// TIA Portal V15.1 export
// export: Created 2024-06-21T08:41:12.1834581Z, ExportSetting WithDefaults, DisplayName Totally Integrated Automation Portal, DisplayVersion V15.1 Update 5, DisplayName TIA Portal Openness, DisplayVersion V15.1 Update 5, DisplayName SINAMICS Startdrive Advanced, DisplayVersion V15.1, DisplayName G130, G150, S120, S150, SINAMICS MV, S210, DisplayVersion V15.1, DisplayName G110M, G120, G120C, G120D, G120P, DisplayVersion V15.1, DisplayName STEP 7 Professional, DisplayVersion V15.1 Update 5, DisplayName STEP 7 Safety, DisplayVersion V15.1, DisplayName WinCC Professional, DisplayVersion V15.1 Update 5, DisplayName SIMATIC Visualization Architect, DisplayVersion V15.1
FUNCTION_BLOCK "LGBShiftRegLineSub"   // FB6705, SCL
TITLE = 'L_ShiftRegLineGC'
{ S7_Optimized_Access := 'TRUE' }
VERSION : 0.1
// Block Parameters
// stored: AutoNumber false, IsIECCheckEnabled false, IsRetainMemResEnabled false, MemoryReserve 100, SetENOAutomatically False, UDAEnableTagReadback false
   VAR_INPUT
      I_VEMData { ExternalAccessible := 'False'; ExternalVisible := 'False'; ExternalWritable := 'False'} : "VEMData";   // VEMData
      I_EncPlsCntr { ExternalAccessible := 'False'; ExternalVisible := 'False'; ExternalWritable := 'False'} : DInt;   // Encoder pulse counter - value from counter card
      I_LineRunning { ExternalAccessible := 'False'; ExternalVisible := 'False'; ExternalWritable := 'False'} : Bool;   // Line running - signal from freq. convertor
      I_TriggerDet { ExternalAccessible := 'False'; ExternalVisible := 'False'; ExternalWritable := 'False'} : Bool;   // Trigger sensor
   END_VAR
   VAR_OUTPUT
      O_SetpBodyPitch { ExternalAccessible := 'False'; ExternalVisible := 'False'; ExternalWritable := 'False'} : Int;   // Setpoint Body pitch (cm)
      O_SetpCycleTime { ExternalAccessible := 'False'; ExternalVisible := 'False'; ExternalWritable := 'False'} : Int;   // Setpoint Cycle time (sec)
      O_SetpSpeed { ExternalAccessible := 'False'; ExternalVisible := 'False'; ExternalWritable := 'False'} : Real;   // Setpoint Speed (m/min)
      O_LineIsEmpty { ExternalAccessible := 'False'; ExternalVisible := 'False'; ExternalWritable := 'False'} : Bool;   // Line is empty
      O_AA_EncoderMinMax { ExternalAccessible := 'False'; ExternalVisible := 'False'; ExternalWritable := 'False'} : Bool;   // Settings Min. and Max. range for the encoder is not ok --- Max. must be > Min. and Max. <> 0
      O_AA_SetpointBodyPitch { ExternalAccessible := 'False'; ExternalVisible := 'False'; ExternalWritable := 'False'} : Bool;   // Setpoint Bodypitch is not ok --- Setpoint must be > 100 cm
      O_AA_SetpointCycleTime { ExternalAccessible := 'False'; ExternalVisible := 'False'; ExternalWritable := 'False'} : Bool;   // Setpoint CycleTime is not ok --- Setpoint must be > 10 sec
      O_AA_NbrOfWorkZones { ExternalAccessible := 'False'; ExternalVisible := 'False'; ExternalWritable := 'False'} : Bool;   // Number of work zones is not ok --- Must be >= 2 and <= 30
      O_AA_EncoderPuls { ExternalAccessible := 'False'; ExternalVisible := 'False'; ExternalWritable := 'False'} : Bool;   // The line is running buth there are no encoder pulses
      O_AC_Calibration { ExternalAccessible := 'False'; ExternalVisible := 'False'; ExternalWritable := 'False'} : Bool;   // Calibration is not ok. Let the line run and start the calibration
      O_AC_Area1 { ExternalAccessible := 'False'; ExternalVisible := 'False'; ExternalWritable := 'False'} : Bool;   // Start or End value is not ok
      O_AC_Area2 { ExternalAccessible := 'False'; ExternalVisible := 'False'; ExternalWritable := 'False'} : Bool;   // Start or End value is not ok
      O_AC_Area3 { ExternalAccessible := 'False'; ExternalVisible := 'False'; ExternalWritable := 'False'} : Bool;   // Start or End value is not ok
      O_AC_Area4 { ExternalAccessible := 'False'; ExternalVisible := 'False'; ExternalWritable := 'False'} : Bool;   // Start or End value is not ok
      O_AC_Area5 { ExternalAccessible := 'False'; ExternalVisible := 'False'; ExternalWritable := 'False'} : Bool;   // Start or End value is not ok
      O_AC_Area6 { ExternalAccessible := 'False'; ExternalVisible := 'False'; ExternalWritable := 'False'} : Bool;   // Start or End value is not ok
      O_AC_Area7 { ExternalAccessible := 'False'; ExternalVisible := 'False'; ExternalWritable := 'False'} : Bool;   // Start or End value is not ok
      O_AC_Area8 { ExternalAccessible := 'False'; ExternalVisible := 'False'; ExternalWritable := 'False'} : Bool;   // Start or End value is not ok
      O_AC_Area9 { ExternalAccessible := 'False'; ExternalVisible := 'False'; ExternalWritable := 'False'} : Bool;   // Start or End value is not ok
      O_AC_Area10 { ExternalAccessible := 'False'; ExternalVisible := 'False'; ExternalWritable := 'False'} : Bool;   // Start or End value is not ok
      O_Area1 { ExternalAccessible := 'False'; ExternalVisible := 'False'; ExternalWritable := 'False'} : Bool;   // Position active in the Area
      O_Area2 { ExternalAccessible := 'False'; ExternalVisible := 'False'; ExternalWritable := 'False'} : Bool;   // Position active in the Area
      O_Area3 { ExternalAccessible := 'False'; ExternalVisible := 'False'; ExternalWritable := 'False'} : Bool;   // Position active in the Area
      O_Area4 { ExternalAccessible := 'False'; ExternalVisible := 'False'; ExternalWritable := 'False'} : Bool;   // Position active in the Area
      O_Area5 { ExternalAccessible := 'False'; ExternalVisible := 'False'; ExternalWritable := 'False'} : Bool;   // Position active in the Area
      O_Area6 { ExternalAccessible := 'False'; ExternalVisible := 'False'; ExternalWritable := 'False'} : Bool;   // Position active in the Area
      O_Area7 { ExternalAccessible := 'False'; ExternalVisible := 'False'; ExternalWritable := 'False'} : Bool;   // Position active in the Area
      O_Area8 { ExternalAccessible := 'False'; ExternalVisible := 'False'; ExternalWritable := 'False'} : Bool;   // Position active in the Area
      O_Area9 { ExternalAccessible := 'False'; ExternalVisible := 'False'; ExternalWritable := 'False'} : Bool;   // Position active in the Area
      O_Area10 { ExternalAccessible := 'False'; ExternalVisible := 'False'; ExternalWritable := 'False'} : Bool;   // Position active in the Area
   END_VAR
   VAR_IN_OUT
      IO_ShiftRegData : "ShiftRegData";   // Line data
      IO_Modes : "Modes";   // Modes
      H_HMI : "H_HMI";   // Animation
      H_GBShiftRegLine : "H_GBShiftRegLine";   // Animation
      C_Config : "ShiftRegLineConfig";   // Config
   END_VAR
   VAR
      AlarmEncoderMinMax { ExternalAccessible := 'False'; ExternalVisible := 'False'; ExternalWritable := 'False'} : Bool;   // Settings Min. and Max. range for the encoder is not ok --- Max. must be > Min. and Max. <> 0
      AlarmSetpointBodyPitch { ExternalAccessible := 'False'; ExternalVisible := 'False'; ExternalWritable := 'False'} : Bool;   // Setpoint Bodypitch is not ok --- Setpoint must be > 100 cm
      AlarmSetpointCycleTime { ExternalAccessible := 'False'; ExternalVisible := 'False'; ExternalWritable := 'False'} : Bool;   // Setpoint CycleTime is not ok --- Setpoint must be > 10 sec
      AlarmNbrOfWorkZones { ExternalAccessible := 'False'; ExternalVisible := 'False'; ExternalWritable := 'False'} : Bool;   // Number of work zones is not ok --- Must be >= 2 and <= 30
      AlarmEncoderPuls { ExternalAccessible := 'False'; ExternalVisible := 'False'; ExternalWritable := 'False'} : Bool;   // The line is running buth there are no encoder pulses
      AlarmCalibration { ExternalAccessible := 'False'; ExternalVisible := 'False'; ExternalWritable := 'False'} : Bool;   // Calibration is not ok. Let the line run and start the calibration
      AlarmArea { ExternalAccessible := 'False'; ExternalVisible := 'False'; ExternalWritable := 'False'} : Array[0..9] of Bool;   // Start or End value is not ok
      AreaPosition { ExternalAccessible := 'False'; ExternalVisible := 'False'; ExternalWritable := 'False'} : Array[0..9] of Bool;   // Position active in the Area
      VEMDataEmpty { ExternalAccessible := 'False'; ExternalVisible := 'False'; ExternalWritable := 'False'} : "VEMData";   // Empty VEMData
      i { ExternalAccessible := 'False'; ExternalVisible := 'False'; ExternalWritable := 'False'} : Int;   // General index
      j { ExternalAccessible := 'False'; ExternalVisible := 'False'; ExternalWritable := 'False'} : Int;   // General index
   END_VAR
   VAR RETAIN
      ZoneNbrMin { ExternalAccessible := 'False'; ExternalVisible := 'False'; ExternalWritable := 'False'} : Int;   // Minimum possible zone - number
      ZoneNbrMax { ExternalAccessible := 'False'; ExternalVisible := 'False'; ExternalWritable := 'False'} : Int;   // Maximum possible zone - number
      EncPlsCntrMem { ExternalAccessible := 'False'; ExternalVisible := 'False'; ExternalWritable := 'False'} : DInt;   // Encoder pulse counter memorized
      EncPlsCntrRngDiv4 { ExternalAccessible := 'False'; ExternalVisible := 'False'; ExternalWritable := 'False'} : DInt;   // Encoder pulse counter range divided by 4
      EncPlsCntr25Pct { ExternalAccessible := 'False'; ExternalVisible := 'False'; ExternalWritable := 'False'} : DInt;   // Encoder pulse counter at 25%
      EncPlsCntr75Pct { ExternalAccessible := 'False'; ExternalVisible := 'False'; ExternalWritable := 'False'} : DInt;   // Encoder pulse counter at 75%
      EncPlsCntrMinOvFlow { ExternalAccessible := 'False'; ExternalVisible := 'False'; ExternalWritable := 'False'} : Bool;   // Encoder pulse counter minimum overflow
      EncPlsCntrMaxOvFlow { ExternalAccessible := 'False'; ExternalVisible := 'False'; ExternalWritable := 'False'} : Bool;   // Encoder pulse counter maximum overflow
      EncPlsCntrDiff { ExternalAccessible := 'False'; ExternalVisible := 'False'; ExternalWritable := 'False'} : DInt;   // Encoder pulse counter difference
      CalibPlsCntr { ExternalAccessible := 'False'; ExternalVisible := 'False'; ExternalWritable := 'False'} : DInt;   // Calibration - pulse counter
      CalibTimAct { ExternalAccessible := 'False'; ExternalVisible := 'False'; ExternalWritable := 'False'} : Real;   // Calibration - actual calibration time
      CalibTimeRemain { ExternalAccessible := 'False'; ExternalVisible := 'False'; ExternalWritable := 'False'} : DInt;   // Calibration - remaining calibration time
      CalibDistTimeRatio { ExternalAccessible := 'False'; ExternalVisible := 'False'; ExternalWritable := 'False'} : Real;   // Calibration temp result
      CalibPlsTimeRatio { ExternalAccessible := 'False'; ExternalVisible := 'False'; ExternalWritable := 'False'} : Real;   // Calibration temp result
      PosDiff { ExternalAccessible := 'False'; ExternalVisible := 'False'; ExternalWritable := 'False'} : Real;   // Position difference - randomized travel distance during 1 or more scans
   END_VAR
   VAR
      LineRampingUp { ExternalAccessible := 'False'; ExternalVisible := 'False'; ExternalWritable := 'False'} : Bool;   // Line ramping up
      LineRampingDown { ExternalAccessible := 'False'; ExternalVisible := 'False'; ExternalWritable := 'False'} : Bool;   // Line ramping down
      StartPos { ExternalAccessible := 'False'; ExternalVisible := 'False'; ExternalWritable := 'False'} : Int;   // Start position
      TriggerDetZone { ExternalAccessible := 'False'; ExternalVisible := 'False'; ExternalWritable := 'False'} : Int;   // Trigger sensor in zone X
      LineDataZoneSelNbr { ExternalAccessible := 'False'; ExternalVisible := 'False'; ExternalWritable := 'False'} : Int;   // Line data zone selection number
      AreaStartPosition { ExternalAccessible := 'False'; ExternalVisible := 'False'; ExternalWritable := 'False'} : Real;   // Area Start Position
      AreaEndPosition { ExternalAccessible := 'False'; ExternalVisible := 'False'; ExternalWritable := 'False'} : Real;   // Area End Position
      SetpointSpeed { ExternalAccessible := 'False'; ExternalVisible := 'False'; ExternalWritable := 'False'} : Real;   // Setpoint speed (m/min)
      ActualSpeed { ExternalAccessible := 'False'; ExternalVisible := 'False'; ExternalWritable := 'False'} : Real;   // Actual speed (m/min)
      SpeedPlsCntr { ExternalAccessible := 'False'; ExternalVisible := 'False'; ExternalWritable := 'False'} : DInt;   // Speed temp result
      SpeedDistRatio { ExternalAccessible := 'False'; ExternalVisible := 'False'; ExternalWritable := 'False'} : Real;   // Speed temp result
      CheckPlsCntrDiffMem { ExternalAccessible := 'False'; ExternalVisible := 'False'; ExternalWritable := 'False'} : DInt;   // Check encoder puls counter - diff between memorized and actual value
      LineIsEmpty { ExternalAccessible := 'False'; ExternalVisible := 'False'; ExternalWritable := 'False'} : Bool;   // Line is empty
      LineRunningForward { ExternalAccessible := 'False'; ExternalVisible := 'False'; ExternalWritable := 'False'} : Bool;   // Line running in forward direction
      LineRunningReverse { ExternalAccessible := 'False'; ExternalVisible := 'False'; ExternalWritable := 'False'} : Bool;   // Line running in reverse direction
      "Pop-upSealing" { ExternalAccessible := 'False'; ExternalVisible := 'False'; ExternalWritable := 'False'} : Bool;   // Show Pop-up Sealing
      "Pop-upPaint" { ExternalAccessible := 'False'; ExternalVisible := 'False'; ExternalWritable := 'False'} : Bool;   // Show Pop-up Paint
      "Pop-upPreTreatment" { ExternalAccessible := 'False'; ExternalVisible := 'False'; ExternalWritable := 'False'} : Bool;   // Show Pop-up Pre-Treatment
      AlarmA { ExternalAccessible := 'False'; ExternalVisible := 'False'; ExternalWritable := 'False'} : Bool;   // Alarm A
      AlarmB { ExternalAccessible := 'False'; ExternalVisible := 'False'; ExternalWritable := 'False'} : Bool;   // Alarm B
      AlarmC { ExternalAccessible := 'False'; ExternalVisible := 'False'; ExternalWritable := 'False'} : Bool;   // Alarm C
      AlarmD { ExternalAccessible := 'False'; ExternalVisible := 'False'; ExternalWritable := 'False'} : Bool;   // Alarm D
      T_LineRampingUP { ExternalAccessible := 'False'; ExternalVisible := 'False'; ExternalWritable := 'False'} : "LTimer";   // TIMER
      T_LineRampingDown { ExternalAccessible := 'False'; ExternalVisible := 'False'; ExternalWritable := 'False'} : "LTimer";   // TIMER
      T_Calibration { ExternalAccessible := 'False'; ExternalVisible := 'False'; ExternalWritable := 'False'} : "LTimer";   // TIMER
      T_SpeedCalculation { ExternalAccessible := 'False'; ExternalVisible := 'False'; ExternalWritable := 'False'} : "LTimer";   // TIMER
      T_AlmEncoderPuls { ExternalAccessible := 'False'; ExternalVisible := 'False'; ExternalWritable := 'False'} : "LTimer";   // TIMER
      F_TRIG_LineRunning { ExternalAccessible := 'False'; ExternalVisible := 'False'; ExternalWritable := 'False'} : F_TRIG;   // TRIGGER
      R_TRIG_LineRunning { ExternalAccessible := 'False'; ExternalVisible := 'False'; ExternalWritable := 'False'} : R_TRIG;   // TRIGGER
      R_TRIG_StartCalibration { ExternalAccessible := 'False'; ExternalVisible := 'False'; ExternalWritable := 'False'} : R_TRIG;   // TRIGGER
      R_TRIG_TriggerDet { ExternalAccessible := 'False'; ExternalVisible := 'False'; ExternalWritable := 'False'} : R_TRIG;   // TRIGGER
      R_TRIG_ZoneOpenClose { ExternalAccessible := 'False'; ExternalVisible := 'False'; ExternalWritable := 'False'} : R_TRIG;   // TRIGGER
      F_TRIG_ZoneDataEdit { ExternalAccessible := 'False'; ExternalVisible := 'False'; ExternalWritable := 'False'} : F_TRIG;   // TRIGGER
      R_TRIG_ZoneDataUpdate { ExternalAccessible := 'False'; ExternalVisible := 'False'; ExternalWritable := 'False'} : R_TRIG;   // TRIGGER
      R_TRIG_ZoneDataDelete { ExternalAccessible := 'False'; ExternalVisible := 'False'; ExternalWritable := 'False'} : R_TRIG;   // TRIGGER
      Comm_ActualPos { ExternalAccessible := 'False'; ExternalVisible := 'False'; ExternalWritable := 'False'} : DInt;
   END_VAR
   VAR_TEMP
      HMICMD : Struct   // Temp
         CalibrationStart : Bool;   // Popup Calibration - Start Calibration
         CallibrationAccept : Bool;   // Popup Calibration - Accept Calibration
         Spare2 : Bool;   // Spare
         Spare3 : Bool;   // Spare
         Spare4 : Bool;   // Spare
         Spare5 : Bool;   // Spare
         Spare6 : Bool;   // Spare
         Spare7 : Bool;   // Spare
         PopupZoneOpenClose : Bool;   // Popup Zone Data - Open / Close
         PopupZoneDataEdit : Bool;   // Popup Zone Data - Edit
         PopupDataUpdate : Bool;   // Popup Zone Data - Update
         PopupDataDelete : Bool;   // Popup Zone Data - Delete
         Spare12 : Bool;   // Spare
         Spare13 : Bool;   // Spare
         Spare14 : Bool;   // Spare
         Spare15 : Bool;   // Spare
         Spare16 : Bool;   // Spare
         Spare17 : Bool;   // Spare
         Spare18 : Bool;   // Spare
         Spare19 : Bool;   // Spare
         Spare20 : Bool;   // Spare
         Spare21 : Bool;   // Spare
         Spare22 : Bool;   // Spare
         Spare23 : Bool;   // Spare
         Spare24 : Bool;   // Spare
         Spare25 : Bool;   // Spare
         Spare26 : Bool;   // Spare
         Spare27 : Bool;   // Spare
         Spare28 : Bool;   // Spare
         Spare29 : Bool;   // Spare
         Spare30 : Bool;   // Spare
         Spare31 : Bool;   // Spare
      END_STRUCT;
   END_VAR
   VAR CONSTANT
      COLOUR_WHITE : Word := 8;
      COLOUR_GREEN : Word := 9;
      COLOUR_YELLOW : Word := 10;
      COLOUR_RED : Word := 11;
   END_VAR
BEGIN
   REGION *** HMI Commands ***
       "LDWordToBit"(I_DWord := #H_HMI.H_CommandDW1,
                     O_0 => #HMICMD.CalibrationStart,
                     O_1 => #HMICMD.CallibrationAccept,
                     O_2 => #HMICMD.Spare2,
                     O_3 => #HMICMD.Spare3,
                     O_4 => #HMICMD.Spare4,
                     O_5 => #HMICMD.Spare5,
                     O_6 => #HMICMD.Spare6,
                     O_7 => #HMICMD.Spare7,
                     O_8 => #HMICMD.PopupZoneOpenClose,
                     O_9 => #HMICMD.PopupZoneDataEdit,
                     O_10 => #HMICMD.PopupDataUpdate,
                     O_11 => #HMICMD.PopupDataDelete,
                     O_12 => #HMICMD.Spare12,
                     O_13 => #HMICMD.Spare13,
                     O_14 => #HMICMD.Spare14,
                     O_15 => #HMICMD.Spare15,
                     O_16 => #HMICMD.Spare16,
                     O_17 => #HMICMD.Spare17,
                     O_18 => #HMICMD.Spare18,
                     O_19 => #HMICMD.Spare19,
                     O_20 => #HMICMD.Spare20,
                     O_21 => #HMICMD.Spare21,
                     O_22 => #HMICMD.Spare22,
                     O_23 => #HMICMD.Spare23,
                     O_24 => #HMICMD.Spare24,
                     O_25 => #HMICMD.Spare25,
                     O_26 => #HMICMD.Spare26,
                     O_27 => #HMICMD.Spare27,
                     O_28 => #HMICMD.Spare28,
                     O_29 => #HMICMD.Spare29,
                     O_30 => #HMICMD.Spare30,
                     O_31 => #HMICMD.Spare31);

   END_REGION

   REGION *** Inputs ***
       #"Pop-upSealing" := False;
       #"Pop-upPaint" := False;
       #"Pop-upPreTreatment" := False;

       IF (#C_Config."Sealing/Paint/PreTreatment" = 1) THEN
           #"Pop-upSealing" := True;
       END_IF;
       IF (#C_Config."Sealing/Paint/PreTreatment" = 2) THEN
           #"Pop-upPaint" := True;
       END_IF;
       IF (#C_Config."Sealing/Paint/PreTreatment" = 3) THEN
           #"Pop-upPreTreatment" := True;
       END_IF;
   END_REGION

   REGION *** Config (for LineFeed FB) *** 

       #IO_ShiftRegData.SetpointBodyPitch := #C_Config.BodyPitch;
       #IO_ShiftRegData.SetpointCycleTime := #C_Config.CycleTime;
       #IO_ShiftRegData.NbrOfWorkZones := #C_Config.NbrOfWorkZones;

   END_REGION

   REGION *** Alarms ***

       //Settings Min. and Max. range for the encoder is not ok --- Max. must be > Min. and Max. <> 0
       #AlarmEncoderMinMax := (#C_Config.EncPlsCntrMin > #C_Config.EncPlsCntrMax) OR (#C_Config.EncPlsCntrMin = #C_Config.EncPlsCntrMax) OR (#C_Config.EncPlsCntrMax = 0);

       //Setpoint Bodypitch is not ok --- Setpoint must be > 100 cm
       #AlarmSetpointBodyPitch := (#C_Config.BodyPitch <= 100);

       //Setpoint CycleTime is not ok --- Setpoint must be > 10 sec
       #AlarmSetpointCycleTime := (#C_Config.CycleTime <= 10);

       //Number of work zones is not ok --- Must be >= 2 and <= 30
       #AlarmNbrOfWorkZones := (#C_Config.NbrOfWorkZones < 2) OR (#C_Config.NbrOfWorkZones > 30);

       //The line is running buth there are no encoder pulses
       #T_AlmEncoderPuls(I_StartTimer := NOT #LineRampingUp AND #I_LineRunning AND NOT #LineRampingDown AND (#EncPlsCntrMem = #I_EncPlsCntr),
                        I_HoldTimer := False,
                        I_MaxTimerValue := 3000,
                        O_TimerResult=>"NotUsedBool",
                        O_TimerValue=>"NotUsedDInt" );

      IF #T_AlmEncoderPuls.O_TimerResult THEN
          #AlarmEncoderPuls := True;
      ELSIF #IO_Modes.LMode.AlarmResetPB THEN
          #AlarmEncoderPuls := FALSE;
      END_IF;

       //Calibration is not ok. Let the line run and start the calibration
      #AlarmCalibration := (#H_GBShiftRegLine.H_PopupCalibrPlsDistRatioAct[1].H_Real <= 0);

       //Start or End value is not ok
       #AlarmArea[0] := #C_Config.Area_Used[0] AND ((#C_Config.Area_EndPosition[0] <= #C_Config.Area_StartPosition[0]) OR (#C_Config.Area_EndPosition[0] > #C_Config.BodyPitch));
       #AlarmArea[1] := #C_Config.Area_Used[1] AND ((#C_Config.Area_EndPosition[1] <= #C_Config.Area_StartPosition[1]) OR (#C_Config.Area_EndPosition[1] > #C_Config.BodyPitch));
       #AlarmArea[2] := #C_Config.Area_Used[2] AND ((#C_Config.Area_EndPosition[2] <= #C_Config.Area_StartPosition[2]) OR (#C_Config.Area_EndPosition[2] > #C_Config.BodyPitch));
       #AlarmArea[3] := #C_Config.Area_Used[3] AND ((#C_Config.Area_EndPosition[3] <= #C_Config.Area_StartPosition[3]) OR (#C_Config.Area_EndPosition[3] > #C_Config.BodyPitch));
       #AlarmArea[4] := #C_Config.Area_Used[4] AND ((#C_Config.Area_EndPosition[4] <= #C_Config.Area_StartPosition[4]) OR (#C_Config.Area_EndPosition[4] > #C_Config.BodyPitch));
       #AlarmArea[5] := #C_Config.Area_Used[5] AND ((#C_Config.Area_EndPosition[5] <= #C_Config.Area_StartPosition[5]) OR (#C_Config.Area_EndPosition[5] > #C_Config.BodyPitch));
       #AlarmArea[6] := #C_Config.Area_Used[6] AND ((#C_Config.Area_EndPosition[6] <= #C_Config.Area_StartPosition[6]) OR (#C_Config.Area_EndPosition[6] > #C_Config.BodyPitch));
       #AlarmArea[7] := #C_Config.Area_Used[7] AND ((#C_Config.Area_EndPosition[7] <= #C_Config.Area_StartPosition[7]) OR (#C_Config.Area_EndPosition[7] > #C_Config.BodyPitch));
       #AlarmArea[8] := #C_Config.Area_Used[8] AND ((#C_Config.Area_EndPosition[8] <= #C_Config.Area_StartPosition[8]) OR (#C_Config.Area_EndPosition[8] > #C_Config.BodyPitch));
       #AlarmArea[9] := #C_Config.Area_Used[9] AND ((#C_Config.Area_EndPosition[9] <= #C_Config.Area_StartPosition[9]) OR (#C_Config.Area_EndPosition[9] > #C_Config.BodyPitch));

   END_REGION

   REGION *** Alarm A/B/C/D ****

       //Alarm A
       #AlarmA := #AlarmEncoderMinMax OR #AlarmSetpointBodyPitch OR #AlarmSetpointCycleTime OR #AlarmNbrOfWorkZones OR #AlarmEncoderPuls;

       //Alarm B
       #AlarmB := False;

       //Alarm C
       #AlarmC := #AlarmCalibration OR #AlarmArea[0] OR #AlarmArea[1] OR #AlarmArea[2] OR #AlarmArea[3] OR #AlarmArea[4] OR #AlarmArea[5] OR #AlarmArea[6] OR #AlarmArea[7] OR #AlarmArea[8] OR #AlarmArea[9];

       //Alarm D
       #AlarmD := False;

   END_REGION

   REGION *** Alarms To Alarm UDT ***

       IF (#AlarmA OR #AlarmB OR #AlarmC OR #AlarmD) AND (#IO_Modes.Alarm.AlarmInstance = WSTRING#'') THEN
           #IO_Modes.Alarm.AlarmInstance := GetInstancePath(0);
       END_IF;

       "LAlarmSummary"(I_AlarmA:= #AlarmA,
                       I_AlarmB:= #AlarmB,
                       I_AlarmC:= #AlarmC,
                       I_AlarmD:= #AlarmD,
                       I_AlarmABCondition:= "FALSE",
                       IO_Alarm:= #IO_Modes.Alarm,
                       C_UpperLevelHW:= "FALSE",
                       C_UpperLevelSafety:= "FALSE",
                       C_Safety:= "FALSE",
                       C_Mechanic:= "FALSE",
                       C_Transport:= "TRUE",
                       C_Feature1:= "FALSE",
                       C_Feature2:= "FALSE",
                       C_Feature3:= "FALSE");

   END_REGION

   REGION *** Line ramping up / down ***

       #R_TRIG_LineRunning(CLK := #I_LineRunning);
       #F_TRIG_LineRunning(CLK := #I_LineRunning);

       IF #R_TRIG_LineRunning.Q THEN
           #LineRampingUp := True;
       END_IF;
       IF #F_TRIG_LineRunning.Q THEN
           #LineRampingDown := True;
       END_IF;

       #T_LineRampingUP(I_StartTimer := #LineRampingUp,
      I_HoldTimer := False,
      I_MaxTimerValue := 5000);
       #T_LineRampingDown(I_StartTimer := #LineRampingDown,
      I_HoldTimer := False,
      I_MaxTimerValue := 5000);

       IF #T_LineRampingUP.O_TimerResult OR NOT #I_LineRunning THEN
           #LineRampingUp := False;
       END_IF;
       IF #T_LineRampingDown.O_TimerResult OR #I_LineRunning THEN
           #LineRampingDown := False;
       END_IF;

   END_REGION

   REGION *** Encoder pulse counter handling ***

       #EncPlsCntrRngDiv4 := #C_Config.EncPlsCntrMax / 4 - #C_Config.EncPlsCntrMin / 4;     //calculate 1/4th of the range
       #EncPlsCntr75Pct := #C_Config.EncPlsCntrMax - #EncPlsCntrRngDiv4;           //75 percent of the encoder counter
       #EncPlsCntr25Pct := #C_Config.EncPlsCntrMin + #EncPlsCntrRngDiv4;           //25 percent of the encoder counter

       IF (#C_Config.EncPlsCntrMax > #C_Config.EncPlsCntrMin) AND (#I_LineRunning OR #LineRampingDown) THEN
           #EncPlsCntrMaxOvFlow := (#I_EncPlsCntr < #EncPlsCntr25Pct) AND (#EncPlsCntrMem > #EncPlsCntr75Pct);
           #EncPlsCntrMinOvFlow := (#I_EncPlsCntr > #EncPlsCntr75Pct) AND (#EncPlsCntrMem < #EncPlsCntr25Pct);

           IF #EncPlsCntrMaxOvFlow THEN
               //Correct pulse counter difference in case of forward flip-over
               #EncPlsCntrDiff := (#C_Config.EncPlsCntrMax - #EncPlsCntrMem) + ROUND_DINT(#I_EncPlsCntr);
           ELSIF #EncPlsCntrMinOvFlow THEN
               //Correct pulse counter difference in case of reverse flip-over
               #EncPlsCntrDiff := ROUND_DINT(#EncPlsCntrMem) + (#C_Config.EncPlsCntrMax - #I_EncPlsCntr);
           ELSE
               #EncPlsCntrDiff := #I_EncPlsCntr - #EncPlsCntrMem;
           END_IF;

           IF #EncPlsCntrDiff > 0 THEN
               //Line running forward
               #LineRunningForward := True;       
               #LineRunningReverse := False;
           ELSIF #EncPlsCntrDiff < 0 THEN
               //Line running reverse
               #LineRunningForward := False;
               #LineRunningReverse := True;       
           END_IF;
       ELSE
             #EncPlsCntrDiff := 0;
             #LineRunningForward := False;
             #LineRunningReverse := False;
       END_IF;

       #EncPlsCntrMem := #I_EncPlsCntr;

   END_REGION

   REGION *** Position difference ***

       #PosDiff := DINT_TO_REAL(#EncPlsCntrDiff) / #H_GBShiftRegLine.H_PopupCalibrPlsDistRatioAct[1].H_Real;

       //Handle sudden jumps in encoder
       IF ABS(#PosDiff) > 10 THEN
           #PosDiff := 0;
       END_IF;

   END_REGION

   REGION *** Line Data -> Position ***

       #ZoneNbrMin := 0;
       #ZoneNbrMax := #C_Config.NbrOfWorkZones + 1;

       IF #ZoneNbrMax > 31 THEN
           #ZoneNbrMax := 31;
       END_IF;

       #StartPos := 0 - #C_Config.BodyPitch;

       FOR #i := 0 TO #ZoneNbrMax DO
           #IO_ShiftRegData.Zone[#i].StartPosition := #StartPos;
           #IO_ShiftRegData.Zone[#i].EndPosition := #StartPos + #C_Config.BodyPitch;
           #IO_ShiftRegData.Zone[#i].Anim.Visible := True;
           #IO_ShiftRegData.Zone[#i].Anim.Freeze := False;
           #IO_ShiftRegData.Zone[#i].Anim.Colour := #COLOUR_WHITE;

           IF (#IO_ShiftRegData.Zone[#i].TagID > 0) THEN
               #IO_ShiftRegData.Zone[#i].ActualPosition := #IO_ShiftRegData.Zone[#i].ActualPosition + #PosDiff;
           END_IF;

           IF (#IO_ShiftRegData.Zone[#i].TagID > 0) AND (#IO_ShiftRegData.Zone[#i].ActualPosition > #IO_ShiftRegData.Zone[#i].EndPosition) THEN
               #IO_ShiftRegData.Zone[#i].Anim.Colour := #COLOUR_RED;
           ELSIF (#IO_ShiftRegData.Zone[#i].TagID > 0) AND (#IO_ShiftRegData.Zone[#i].ActualPosition <= #IO_ShiftRegData.Zone[#i].EndPosition) THEN
               #IO_ShiftRegData.Zone[#i].Anim.Colour := #COLOUR_GREEN;
           END_IF;

           #StartPos := #StartPos + #C_Config.BodyPitch;
       END_FOR;

       //Clear the zones which are not used
       FOR #i := #ZoneNbrMax + 1 TO 31 DO
           #IO_ShiftRegData.Zone[#i].TagID := 0;
           #IO_ShiftRegData.Zone[#i].ActualPosition := 0.0;
           #IO_ShiftRegData.Zone[#i].StartPosition := 0.0;
           #IO_ShiftRegData.Zone[#i].EndPosition := 0.0;
           #IO_ShiftRegData.Zone[#i].Anim.Visible := False;
           #IO_ShiftRegData.Zone[#i].Anim.Freeze := False;
           #IO_ShiftRegData.Zone[#i].Anim.Colour := 0;
           #IO_ShiftRegData.Zone[#i].VEMData := #VEMDataEmpty;
       END_FOR;

   END_REGION

   REGION *** Actual bodypitch ***

       #i := 1;
       WHILE #IO_ShiftRegData.Zone[#i].TagID = 0 AND #i < #ZoneNbrMax DO
           #i := #i + 1;
       END_WHILE;

       IF #i = #ZoneNbrMax THEN
           #IO_ShiftRegData.ActualBodyPitch := INT_TO_REAL(#C_Config.BodyPitch);
           #IO_ShiftRegData.ActualBodyPitchZoneX := INT_TO_REAL(#C_Config.BodyPitch);
       ELSE
           #IO_ShiftRegData.ActualBodyPitch := #IO_ShiftRegData.Zone[#i].ActualPosition - DINT_TO_REAL(#C_Config.InfeedConvStopDetPosition);
           #IO_ShiftRegData.ActualBodyPitchZoneX := #IO_ShiftRegData.Zone[#i].ActualPosition - ((#i * INT_TO_REAL(#C_Config.BodyPitch)) - INT_TO_REAL(#C_Config.BodyPitch)) - DINT_TO_REAL(#C_Config.InfeedConvStopDetPosition);
       END_IF;

   END_REGION

   REGION *** Trigger sensor ***

       #R_TRIG_TriggerDet(CLK:=#I_TriggerDet);

       //Trigger sensor - Calculate sensor zone
       IF #C_Config.TriggerDetPosition < 0 THEN
           #TriggerDetZone := 0;
       ELSE
           #TriggerDetZone := (DINT_TO_INT(#C_Config.TriggerDetPosition) / #C_Config.BodyPitch) + 1;
       END_IF;

       //Trigger sensor - Fill in temporary mixnumber in zone 0
       IF #R_TRIG_TriggerDet.Q THEN
           #IO_ShiftRegData.Zone[#TriggerDetZone].TagID := #I_VEMData.Identification;
           #IO_ShiftRegData.Zone[#TriggerDetZone].VEMData := #I_VEMData;
           #IO_ShiftRegData.Zone[#TriggerDetZone].ActualPosition := #C_Config.TriggerDetPosition;
       END_IF;

   END_REGION

   REGION *** Shift data forward ***

       IF #LineRunningForward THEN

           FOR #i := #ZoneNbrMax TO 0 BY -1 DO

               IF #i = #ZoneNbrMax THEN
                   IF (#IO_ShiftRegData.Zone[#i].ActualPosition >= #IO_ShiftRegData.Zone[#i].EndPosition) THEN
                       #IO_ShiftRegData.Zone[#i].TagID := 0;
                       #IO_ShiftRegData.Zone[#i].VEMData := #VEMDataEmpty;
                       #IO_ShiftRegData.Zone[#i].ActualPosition := 0.0;
                   END_IF;
               ELSE
                   IF (#IO_ShiftRegData.Zone[#i].ActualPosition >= #IO_ShiftRegData.Zone[#i].EndPosition) AND (#IO_ShiftRegData.Zone[#i + 1].TagID = 0) THEN
                       #IO_ShiftRegData.Zone[#i + 1].ActualPosition := #IO_ShiftRegData.Zone[#i].ActualPosition;
                       #IO_ShiftRegData.Zone[#i + 1].TagID := #IO_ShiftRegData.Zone[#i].TagID;
                       #IO_ShiftRegData.Zone[#i + 1].VEMData := #IO_ShiftRegData.Zone[#i].VEMData;
                       #IO_ShiftRegData.Zone[#i].TagID := 0;
                       #IO_ShiftRegData.Zone[#i].VEMData := #VEMDataEmpty;
                       #IO_ShiftRegData.Zone[#i].ActualPosition := 0.0;
                   END_IF;
               END_IF;

           END_FOR;
       END_IF;

   END_REGION

   REGION *** Shift data reverse ***

       IF #LineRunningReverse THEN

           FOR #i := 1 TO #ZoneNbrMax BY 1 DO

               IF #i = 1 THEN
                   IF (#IO_ShiftRegData.Zone[#i].ActualPosition < #IO_ShiftRegData.Zone[#i].StartPosition) THEN
                       #IO_ShiftRegData.Zone[0].TagID := #IO_ShiftRegData.Zone[#i].TagID;
                       #IO_ShiftRegData.Zone[0].VEMData := #IO_ShiftRegData.Zone[#i].VEMData;
                       #IO_ShiftRegData.Zone[0].ActualPosition := #IO_ShiftRegData.Zone[#i].ActualPosition;
                       #IO_ShiftRegData.Zone[#i].TagID := 0;
                       #IO_ShiftRegData.Zone[#i].VEMData := #VEMDataEmpty;
                       #IO_ShiftRegData.Zone[#i].ActualPosition := 0.0;
                   END_IF;
               ELSE
                   IF (#IO_ShiftRegData.Zone[#i].ActualPosition < #IO_ShiftRegData.Zone[#i].StartPosition) AND (#IO_ShiftRegData.Zone[#i - 1].TagID = 0) THEN
                       #IO_ShiftRegData.Zone[#i - 1].ActualPosition := #IO_ShiftRegData.Zone[#i].ActualPosition;
                       #IO_ShiftRegData.Zone[#i - 1].TagID := #IO_ShiftRegData.Zone[#i].TagID;
                       #IO_ShiftRegData.Zone[#i - 1].VEMData := #IO_ShiftRegData.Zone[#i].VEMData;
                       #IO_ShiftRegData.Zone[#i].TagID := 0;
                       #IO_ShiftRegData.Zone[#i].VEMData := #VEMDataEmpty;
                       #IO_ShiftRegData.Zone[#i].ActualPosition := 0.0;
                   END_IF;
               END_IF;

           END_FOR;
       END_IF;

   END_REGION

   REGION *** Part Present ***

       FOR #i := #ZoneNbrMax TO 0 BY -1 DO

           IF #IO_ShiftRegData.Zone[#i].TagID <> 0 THEN
               #IO_ShiftRegData.Zone[#i].PartPresent := TRUE;
           ELSE
               #IO_ShiftRegData.Zone[#i].PartPresent := FALSE;
           END_IF;

       END_FOR;

   END_REGION

   REGION *** Line is Empty ***

       #LineIsEmpty := True;
       FOR #i := #ZoneNbrMax TO 0 BY -1 DO

           IF #IO_ShiftRegData.Zone[#i].PartPresent THEN
               #LineIsEmpty := False;
           END_IF;

       END_FOR;

       #IO_ShiftRegData.LineIsEmpty := #LineIsEmpty;

   END_REGION

   REGION *** Line is Running ***

       IF (#ActualSpeed > 0.0) THEN
           #IO_ShiftRegData.LineIsRunning := True;
       ELSE
           #IO_ShiftRegData.LineIsRunning := False;
       END_IF;

   END_REGION

   REGION *** AREA positios ***

       FOR #i := 0 TO 9 BY 1 DO

           #AreaStartPosition := 0;
           #AreaEndPosition := 0;
           #AreaPosition[#i] := False;
           IF #C_Config.Area_Used[#i] THEN
               #j := #C_Config.Area_InZoneX[#i];
               #AreaStartPosition := INT_TO_REAL(#C_Config.Area_StartPosition[#i]) + #IO_ShiftRegData.Zone[#j].StartPosition;
               #AreaEndPosition := INT_TO_REAL(#C_Config.Area_EndPosition[#i]) + #IO_ShiftRegData.Zone[#j].StartPosition;
               IF (#AreaStartPosition < #AreaEndPosition) AND (#AreaStartPosition >=0) THEN
                   IF (#IO_ShiftRegData.Zone[#j].ActualPosition > #AreaStartPosition) AND (#IO_ShiftRegData.Zone[#j].ActualPosition < #AreaEndPosition) THEN
                       #AreaPosition[#i] := True;
                   END_IF;
                   #H_GBShiftRegLine.H_AreaStartPosition[#i].H_DInt := REAL_TO_DINT(#AreaStartPosition);
                   #H_GBShiftRegLine.H_AreaEndPosition[#i].H_DInt := REAL_TO_DINT(#AreaEndPosition);
               ELSE
                   #H_GBShiftRegLine.H_AreaStartPosition[#i].H_DInt := 0;
                   #H_GBShiftRegLine.H_AreaEndPosition[#i].H_DInt := 0;
               END_IF;
           END_IF;
           IF NOT #C_Config.Area_Used[#i] THEN
               #H_GBShiftRegLine.H_AreaStartPosition[#i].H_DInt := 0;
               #H_GBShiftRegLine.H_AreaEndPosition[#i].H_DInt := 0;
           END_IF;

           // Icon Animation
           "LIAnimDWord"(I_SetPos := #AreaPosition[#i],
                         I_ResetPos := FALSE,
                         I_Active := FALSE,
                         I_Visible := TRUE,
                         I_OutOfUse := NOT #C_Config.Area_Used[#i],
                         I_IntlkSet := FALSE,
                         I_IntlkReset := FALSE,
                         I_IntlkSetAlm := FALSE,
                         I_IntlkResetAlm := FALSE,
                         I_ManualMode := FALSE,
                         I_FncSelInHMI := FALSE,
                         I_AnySelected := FALSE,
                         I_AlarmA := FALSE,
                         I_AlarmB := FALSE,
                         I_AlarmC := #AlarmArea[#i],
                         I_AlarmD := FALSE,
                         I_SafetyOk := FALSE,
                         I_Service := FALSE,
                         I_Spare1 := FALSE,
                         I_Spare2 := FALSE,
                         I_Spare3 := FALSE,
                         I_Spare4 := FALSE,
                         I_Spare5 := FALSE,
                         I_Spare6 := FALSE,
                         I_Spare7 := FALSE,
                         I_Spare8 := FALSE,
                         I_Spare9 := FALSE,
                         I_Spare10 := FALSE,
                         I_Spare11 := FALSE,
                         I_Spare12 := FALSE,
                         I_Spare13 := FALSE,
                         I_Spare14 := FALSE,
                         H_IAnim => #H_GBShiftRegLine.H_AreaIAnim[#i].H_DWord);

           // HMI                
           #H_GBShiftRegLine.H_AreaInZoneX[#i].H_Int := #C_Config.Area_InZoneX[#i];

       END_FOR;

   END_REGION

   REGION *** Calibration ***

       #R_TRIG_StartCalibration(CLK := #HMICMD.CalibrationStart);

       //Start calibration timer        
       IF #R_TRIG_StartCalibration.Q THEN
           #CalibPlsCntr := 0;
       ELSIF #HMICMD.CalibrationStart THEN
           #CalibPlsCntr := #CalibPlsCntr + #EncPlsCntrDiff;
       END_IF;

       #T_Calibration(I_StartTimer := #HMICMD.CalibrationStart,
                      I_HoldTimer := false,
                      I_MaxTimerValue := 60000);
       #CalibTimeRemain := (60000 - #T_Calibration.O_TimerValue) / 1000;

       IF #HMICMD.CalibrationStart THEN
           #CalibTimAct := DINT_TO_REAL(#T_Calibration.O_TimerValue) / 1000;
           #CalibDistTimeRatio := INT_TO_REAL(#C_Config.BodyPitch) / INT_TO_REAL(#C_Config.CycleTime);
           #CalibPlsTimeRatio := DINT_TO_REAL(#CalibPlsCntr) / #CalibTimAct;
           #H_GBShiftRegLine.H_PopupCalibrPlsDistRatioNew[1].H_Real := #CalibPlsTimeRatio / #CalibDistTimeRatio;
       END_IF;
       IF #T_Calibration.O_TimerResult THEN
           #H_HMI.H_CommandDW1.%X0 := FALSE;
       END_IF;

       //Use pulse distance ratio from calibration
       IF #HMICMD.CallibrationAccept THEN
           #H_GBShiftRegLine.H_PopupCalibrPlsDistRatioAct[1].H_Real := #H_GBShiftRegLine.H_PopupCalibrPlsDistRatioNew[1].H_Real;
           #H_HMI.H_CommandDW1.%X1 := FALSE;
       END_IF;

       // HMI
       #H_GBShiftRegLine.H_PopupCalibrTimeRemaining[1].H_Int := DINT_TO_INT(#CalibTimeRemain);

   END_REGION

   REGION *** Pop-up Data Edit/Update/Delete ***

       #R_TRIG_ZoneOpenClose(CLK := #HMICMD.PopupZoneOpenClose);
       #F_TRIG_ZoneDataEdit(CLK := #HMICMD.PopupZoneDataEdit);
       #R_TRIG_ZoneDataUpdate(CLK := #HMICMD.PopupDataUpdate);
       #R_TRIG_ZoneDataDelete(CLK := #HMICMD.PopupDataDelete);

       // OPEN Popup OR Deactived EDIT by button without UPDATE or DELETE function
       #i := #H_GBShiftRegLine.H_LineDataZoneDetailNbr[#H_GBShiftRegLine.H_PopupZoneDataSelNbr[1].H_Int].H_Int;
       IF #R_TRIG_ZoneOpenClose.Q OR #F_TRIG_ZoneDataEdit.Q THEN
           #H_GBShiftRegLine.H_PopupZoneDataSelZone[1].H_Int := #i;
           #H_GBShiftRegLine.H_PopupZoneDataSelTagID[1].H_UDInt := #IO_ShiftRegData.Zone[#i].TagID;
           #H_GBShiftRegLine.H_PopupZoneDataSelVemData[1] := #IO_ShiftRegData.Zone[#i].VEMData;
           #H_GBShiftRegLine.H_PopupZoneDataSelPosition[1].H_DInt := REAL_TO_DINT(#IO_ShiftRegData.Zone[#i].ActualPosition);
           #H_HMI.H_CommandDW1.%X8 := FALSE;
           #H_HMI.H_CommandDW1.%X9 := FALSE;
           #H_HMI.H_CommandDW1.%X10 := FALSE;
           #H_HMI.H_CommandDW1.%X11 := FALSE;
       END_IF;

       // UPDATE
       IF #R_TRIG_ZoneDataUpdate.Q THEN
           #IO_ShiftRegData.Zone[#i].VEMData := #H_GBShiftRegLine.H_PopupZoneDataSelVemData[1];
           #H_GBShiftRegLine.H_PopupZoneDataSelTagID[1].H_UDInt := #H_GBShiftRegLine.H_PopupZoneDataSelVemData[1].Identification;
           #IO_ShiftRegData.Zone[#i].TagID := #H_GBShiftRegLine.H_PopupZoneDataSelVemData[1].Identification;
           #IO_ShiftRegData.Zone[#i].ActualPosition := DINT_TO_REAL(#H_GBShiftRegLine.H_PopupZoneDataSelPosition[1].H_DInt);
           #H_HMI.H_CommandDW1.%X9 := FALSE;
           #H_HMI.H_CommandDW1.%X10 := FALSE;
       END_IF;

       // DELETE
       IF #R_TRIG_ZoneDataDelete.Q THEN
           #H_GBShiftRegLine.H_PopupZoneDataSelTagID[1].H_UDInt := 0;
           #H_GBShiftRegLine.H_PopupZoneDataSelVemData[1] := #VEMDataEmpty;
           #H_GBShiftRegLine.H_PopupZoneDataSelPosition[1].H_DInt := 0;
           #IO_ShiftRegData.Zone[#i].TagID := 0;
           #IO_ShiftRegData.Zone[#i].VEMData := #VEMDataEmpty;
           #IO_ShiftRegData.Zone[#i].ActualPosition := 0.0;
           #H_HMI.H_CommandDW1.%X9 := FALSE;
           #H_HMI.H_CommandDW1.%X11 := FALSE;
       END_IF;

   END_REGION

   REGION *** Speed ***

       // Setpoint
       IF (#C_Config.CycleTime <> 0) AND (#C_Config.BodyPitch <> 0) THEN
           #SetpointSpeed := (60.0 / INT_TO_REAL(#C_Config.CycleTime)) * (INT_TO_REAL(#C_Config.BodyPitch) / 100.0);
         ELSE
           #SetpointSpeed := 0.0;
       END_IF;

       // Actual
       #T_SpeedCalculation(I_StartTimer := #I_LineRunning AND NOT #LineRampingUp AND NOT #T_SpeedCalculation.O_TimerResult,
                          I_HoldTimer := False,
                          I_MaxTimerValue := 10000);

      IF #I_LineRunning AND NOT #LineRampingUp THEN
          #SpeedPlsCntr := #SpeedPlsCntr + #EncPlsCntrDiff;
      ELSE
          #SpeedPlsCntr := 0;
      END_IF;

      IF #T_SpeedCalculation.O_TimerResult THEN
          #SpeedDistRatio := DINT_TO_REAL(#SpeedPlsCntr) / #H_GBShiftRegLine.H_PopupCalibrPlsDistRatioAct[1].H_Real;
          #ActualSpeed := 6.0 * (#SpeedDistRatio / 100.0);
          #SpeedPlsCntr := 0;
      END_IF;

   END_REGION

   REGION *** Outputs ***

       #O_SetpBodyPitch := #H_GBShiftRegLine.H_SetpointBodyPitch[1].H_Int;
       #O_SetpCycleTime := #H_GBShiftRegLine.H_SetpointCycleTime[1].H_Int;
       #O_SetpSpeed := #H_GBShiftRegLine.H_SetpointSpeed[1].H_Real;
       #O_LineIsEmpty := #LineIsEmpty;

       #O_AA_EncoderMinMax := #AlarmEncoderMinMax;
       #O_AA_SetpointBodyPitch := #AlarmSetpointBodyPitch;
       #O_AA_SetpointCycleTime := #AlarmSetpointCycleTime;
       #O_AA_NbrOfWorkZones := #AlarmNbrOfWorkZones;
       #O_AA_EncoderPuls := #AlarmEncoderPuls;
       #O_AC_Calibration := #AlarmCalibration;
       #O_AC_Area1 := #AlarmArea[0];
       #O_AC_Area2 := #AlarmArea[1];
       #O_AC_Area3 := #AlarmArea[2];
       #O_AC_Area4 := #AlarmArea[3];
       #O_AC_Area5 := #AlarmArea[4];
       #O_AC_Area6 := #AlarmArea[5];
       #O_AC_Area7 := #AlarmArea[6];
       #O_AC_Area8 := #AlarmArea[7];
       #O_AC_Area9 := #AlarmArea[8];
       #O_AC_Area10 := #AlarmArea[9];

       #O_Area1 := #AreaPosition[0];
       #O_Area2 := #AreaPosition[1];
       #O_Area3 := #AreaPosition[2];
       #O_Area4 := #AreaPosition[3];
       #O_Area5 := #AreaPosition[4];
       #O_Area6 := #AreaPosition[5];
       #O_Area7 := #AreaPosition[6];
       #O_Area8 := #AreaPosition[7];
       #O_Area9 := #AreaPosition[8];
       #O_Area10 := #AreaPosition[9];

   END_REGION

   REGION *** HMI ***

       REGION *** Values ***

           FOR #i := 0 TO 31 BY 1 DO
               #H_GBShiftRegLine.H_LineDataZoneAnim[#i].H_Word := #IO_ShiftRegData.Zone[#i].Anim.Colour;
           END_FOR;

           #LineDataZoneSelNbr := #H_GBShiftRegLine.H_LineDataZoneSelNbr[1].H_Int;
           FOR #i := 0 TO 7 BY 1 DO
               IF #LineDataZoneSelNbr <= #ZoneNbrMax THEN
                   #H_GBShiftRegLine.H_LineDataZoneDetailNbr[#i].H_Int := #LineDataZoneSelNbr;
                   #H_GBShiftRegLine.H_LineDataZoneDetailTagID[#i].H_UDInt := #IO_ShiftRegData.Zone[#LineDataZoneSelNbr].TagID;
                   #H_GBShiftRegLine.H_LineDataZoneDetailVemData[#i] := #IO_ShiftRegData.Zone[#LineDataZoneSelNbr].VEMData;
                   #H_GBShiftRegLine.H_LineDataZoneDetailPosition[#i].H_DInt := REAL_TO_DINT(#IO_ShiftRegData.Zone[#LineDataZoneSelNbr].ActualPosition);
                   #H_GBShiftRegLine.H_LineDataZoneDetailStartPosition[#i].H_DInt := REAL_TO_DINT(#IO_ShiftRegData.Zone[#LineDataZoneSelNbr].StartPosition);
                   #H_GBShiftRegLine.H_LineDataZoneDetailAnim[#i].H_Word := #IO_ShiftRegData.Zone[#LineDataZoneSelNbr].Anim.Colour;
               END_IF;
               IF #LineDataZoneSelNbr > #ZoneNbrMax THEN
                   #H_GBShiftRegLine.H_LineDataZoneDetailNbr[#i].H_Int := 0;
                   #H_GBShiftRegLine.H_LineDataZoneDetailTagID[#i].H_UDInt := 0;
                   #H_GBShiftRegLine.H_LineDataZoneDetailVemData[#i] := #VEMDataEmpty;
                   #H_GBShiftRegLine.H_LineDataZoneDetailPosition[#i].H_DInt := 0;
                   #H_GBShiftRegLine.H_LineDataZoneDetailStartPosition[#i].H_DInt := 0;
                   #H_GBShiftRegLine.H_LineDataZoneDetailAnim[#i].H_Word := 0;
               END_IF;
               #LineDataZoneSelNbr := #LineDataZoneSelNbr + 1;
           END_FOR;
           #Comm_ActualPos := REAL_TO_DINT(#IO_ShiftRegData.Zone[1].ActualPosition);
           #H_GBShiftRegLine.H_ActualBodyPitch[1].H_Int := REAL_TO_INT(#IO_ShiftRegData.ActualBodyPitch);
           #H_GBShiftRegLine.H_SetpointBodyPitch[1].H_Int := #C_Config.BodyPitch;
           #H_GBShiftRegLine.H_SetpointCycleTime[1].H_Int := #C_Config.CycleTime;
           #H_GBShiftRegLine.H_ActualSpeed[1].H_Real := #ActualSpeed;
           #H_GBShiftRegLine.H_SetpointSpeed[1].H_Real := #SetpointSpeed;
           #H_GBShiftRegLine.H_LengthProductionLine[1].H_Int := #C_Config.BodyPitch * #C_Config.NbrOfWorkZones;
           #H_GBShiftRegLine.H_NbrOfWorkZones[1].H_Int := #C_Config.NbrOfWorkZones;
           #H_GBShiftRegLine.H_TriggerDetPosition[1].H_DInt := #C_Config.TriggerDetPosition;
           #H_GBShiftRegLine.H_InfeedConvStopDetPosition[1].H_DInt := #C_Config.InfeedConvStopDetPosition;

       END_REGION;

       REGION *** Animations ***

           "LBitToDword"(I_0 := #AlarmEncoderMinMax,
                         I_1 := #AlarmSetpointBodyPitch,
                         I_2 := #AlarmSetpointCycleTime,
                         I_3 := #AlarmNbrOfWorkZones,
                         I_4 := #AlarmEncoderPuls,
                         I_5 := #AlarmCalibration,
                         I_6 := FALSE,
                         I_7 := FALSE,
                         I_8 := FALSE,
                         I_9 := FALSE,
                         I_10 := #"Pop-upSealing",
                         I_11 := #"Pop-upPaint",
                         I_12 := #"Pop-upPreTreatment",
                         I_13 := FALSE,
                         I_14 := FALSE,
                         I_15 := FALSE,
                         I_16 := #IO_Modes.LMode.ManualMode,
                         I_17 := #IO_Modes.LMode.ManualMode AND #H_HMI.H_CommandDW1.%X9,
                         I_18 := #IO_Modes.LMode.ManualMode AND #H_HMI.H_CommandDW1.%X9,
                         I_19 := #H_HMI.H_CommandDW1.%X0,
                         I_20 := FALSE,
                         I_21 := FALSE,
                         I_22 := FALSE,
                         I_23 := FALSE,
                         I_24 := FALSE,
                         I_25 := FALSE,
                         I_26 := FALSE,
                         I_27 := FALSE,
                         I_28 := FALSE,
                         I_29 := FALSE,
                         I_30 := FALSE,
                         I_31 := FALSE,
                         O_DWord => #H_GBShiftRegLine.H_Anim[1].H_DWord);

       END_REGION

       REGION *** Icon Animation ***

           "LIAnimDWord"(I_SetPos := FALSE,
                         I_ResetPos := FALSE,
                         I_Active := NOT #LineIsEmpty,
                         I_Visible := FALSE,
                         I_OutOfUse := FALSE,
                         I_IntlkSet := FALSE,
                         I_IntlkReset := FALSE,
                         I_IntlkSetAlm := FALSE,
                         I_IntlkResetAlm := FALSE,
                         I_ManualMode := FALSE,
                         I_FncSelInHMI := FALSE,
                         I_AnySelected := FALSE,
                         I_AlarmA := #AlarmA,
                         I_AlarmB := #AlarmB,
                         I_AlarmC := #AlarmC,
                         I_AlarmD := #AlarmD,
                         I_SafetyOk := FALSE,
                         I_Service := FALSE,
                         I_Spare1 := FALSE,
                         I_Spare2 := FALSE,
                         I_Spare3 := FALSE,
                         I_Spare4 := FALSE,
                         I_Spare5 := FALSE,
                         I_Spare6 := FALSE,
                         I_Spare7 := FALSE,
                         I_Spare8 := FALSE,
                         I_Spare9 := FALSE,
                         I_Spare10 := FALSE,
                         I_Spare11 := FALSE,
                         I_Spare12 := FALSE,
                         I_Spare13 := FALSE,
                         I_Spare14 := FALSE,
                         H_IAnim => #H_HMI.H_IAnim);

           "LIAnimDWord"(I_SetPos := FALSE,
                         I_ResetPos := FALSE,
                         I_Active := FALSE,
                         I_Visible := FALSE,
                         I_OutOfUse := FALSE,
                         I_IntlkSet := FALSE,
                         I_IntlkReset := FALSE,
                         I_IntlkSetAlm := FALSE,
                         I_IntlkResetAlm := FALSE,
                         I_ManualMode := FALSE,
                         I_FncSelInHMI := FALSE,
                         I_AnySelected := FALSE,
                         I_AlarmA := #AlarmEncoderPuls,
                         I_AlarmB := FALSE,
                         I_AlarmC := FALSE,
                         I_AlarmD := FALSE,
                         I_SafetyOk := FALSE,
                         I_Service := FALSE,
                         I_Spare1 := FALSE,
                         I_Spare2 := FALSE,
                         I_Spare3 := FALSE,
                         I_Spare4 := FALSE,
                         I_Spare5 := FALSE,
                         I_Spare6 := FALSE,
                         I_Spare7 := FALSE,
                         I_Spare8 := FALSE,
                         I_Spare9 := FALSE,
                         I_Spare10 := FALSE,
                         I_Spare11 := FALSE,
                         I_Spare12 := FALSE,
                         I_Spare13 := FALSE,
                         I_Spare14 := FALSE,
                         H_IAnim => #H_GBShiftRegLine.H_EncoderIAnim[1].H_DWord);

       END_REGION

   END_REGION
END_FUNCTION_BLOCK
